FUNCTION_BLOCK LinearAxis EXTENDS SM_LinearAxis;
VAR_INPUT
END_VAR
VAR_OUTPUT
END_VAR
VAR
    _testVar_LinearAxis : BOOL;
END_VAR

SUPER^();

END_FUNCTION_BLOCK

(* stored: Version 1.1.0.1, ProductVersion 3.1.4018.2
   POU LinearAxis: Id {eb39d377-f253-4d60-9db3-aa3565f100db}, SpecialFunc None *)
